// TIA Portal V17 export
// export: Created 2023-12-05T13:40:23.029701Z, ExportSetting WithDefaults, DisplayName Totally Integrated Automation Portal, DisplayVersion V17, DisplayName TIA Portal Openness, DisplayVersion V17, DisplayName TIA Portal Version Control Interface, DisplayVersion V17, DisplayName SINAMICS Startdrive Advanced, DisplayVersion V17, DisplayName SINAMICS Startdrive G130, G150, S120, S150, SINAMICS MV, S210, DisplayVersion V17, DisplayName SINAMICS Startdrive G110M, G120, G120C, G120D, G120P, G115D, DisplayVersion V17, DisplayName STEP 7 Professional, DisplayVersion V17, DisplayName STEP 7 Safety, DisplayVersion V17, DisplayName WinCC Professional, DisplayVersion V17
FUNCTION "FC532 ACWN_V5_1_7 Alarms" : Void   // FC532, LAD
{ S7_Optimized_Access := 'TRUE' }
VERSION : 0.1
// LG 25.04.2023 => Changed name of the block and structures for STD BLCK V5.1.7
// stored: AutoNumber false, IsIECCheckEnabled false, SetENOAutomatically false, UDAEnableTagReadback false
   VAR_INPUT
      AckStep : Bool;
      "SB DB" : Int;
      "Alarm DB" : Int;
      "Alarm Offset" : Int;
   END_VAR
   VAR_TEMP
      "SB DBW" : Word;
      "AL DBW" : Word;
      "TR DBW" : Word;
   END_VAR
BEGIN

NETWORK
TITLE = Initialization
      L     #"SB DB";
      T     #"SB DBW";
      L     #"Alarm DB";
      T     #"AL DBW";
      L     #"Alarm Offset";
      SLD   3;
      LAR1;

NETWORK
TITLE = Cylinder faults
      CLR;
      OPN   DB [#"SB DBW"];
      L     %DBW72;
      OPN   DB [#"AL DBW"];
      T     DBW [AR1, P#0.0];

NETWORK
TITLE = RCFaults
      A     #AckStep;
      JCN   eno;
      CLR;
      OPN   DB [#"SB DBW"];
      L     %DBB76;
      OPN   DB [#"AL DBW"];
      T     DBB [AR1, P#4.0];
eno:  NOP   0;

NETWORK
TITLE = Faults .0
      CLR;
      OPN   DB [#"SB DBW"];
      A     %DBX78.0;
      OPN   DB [#"AL DBW"];
      =     DBX [AR1, P#5.5];

NETWORK
TITLE = Faults .2
      CLR;
      OPN   DB [#"SB DBW"];
      A     %DBX78.2;
      OPN   DB [#"AL DBW"];
      =     DBX [AR1, P#5.7];

NETWORK
TITLE = Faults .3
      CLR;
      OPN   DB [#"SB DBW"];
      A     %DBX78.3;
      OPN   DB [#"AL DBW"];
      =     DBX [AR1, P#6.0];

NETWORK
TITLE = Faults .4
      CLR;
      OPN   DB [#"SB DBW"];
      A     %DBX78.4;
      OPN   DB [#"AL DBW"];
      =     DBX [AR1, P#6.1];
END_FUNCTION
